PROGRAM PRG_04_SawAxes
VAR
	bUP						: BOOL;
	bDOWN					: BOOL;
	bCUT					: BOOL;
	bRETURN					: BOOL;
	
	bDoublePassCountUp		: BOOL;
	
	ctu_DoublePass			: CTU;
	
	iStep: INT;
	bUP_TON: TON;
//	bUP_TP: TP;
	rtrig1: r_trig;
//	ftrig1: f_trig;
	DoublePass_SR: SR;
	bDoublePassQ: BOOL;
	bUP_TON_IN: BOOL;
	autocrosscut_error: TON;
	RS_TriggerReturn: RS;
	RS_TriggerCUT: RS;
	R_TRIG_0: R_TRIG;
	R_TRIG_1: R_TRIG;
	R_TRIG_2: R_TRIG;
	R_TRIG_3: R_TRIG;
	R_TRIG_4: R_TRIG;
	R_TRIG_5: R_TRIG;
	RS_TriggerCUT2: RS;
	R_TRIG_10: R_TRIG;
	R_TRIG_11: R_TRIG;
	R_TRIG_12: R_TRIG;
	RS_TriggerReturn2: RS;
	R_TRIG_13: R_TRIG;
	R_TRIG_14: R_TRIG;
	R_TRIG_15: R_TRIG;

	rCutSpeed: REAL;
	rReturnSpeed: REAL;
	rVFDMaxSpeed: REAL;
	rBufferSpeed: REAL;
	rSawOFFSpeed: REAL;
	rSpeedScaled: REAL;
	// speed test
	iSpeedTest: INT;
	rSawCurrentTest: REAL;
	TON_step10: TON;
	TON_step20: TON;
	TON_step30: TON;
	TON_step40: TON;
	TON_step50: TON;
	TON_step60: TON;
	TON_DownDelay: TON;
END_VAR

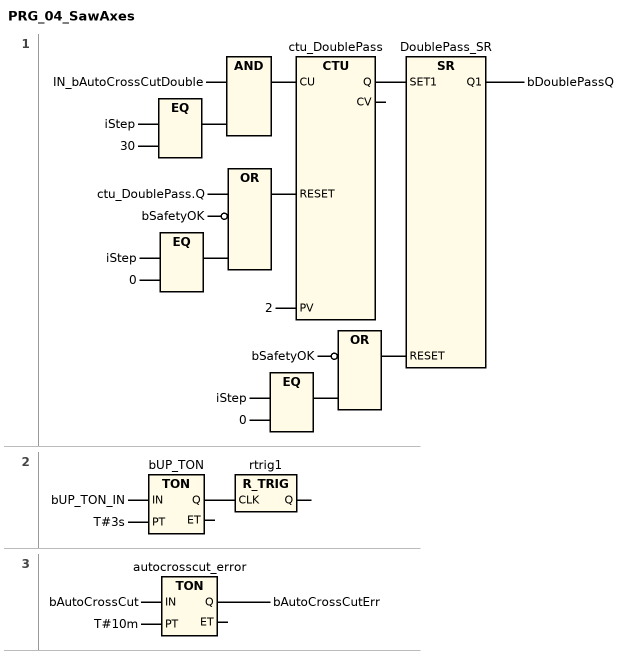
// NETWORK 1
ctu_DoublePass(
    CU := IN_bAutoCrossCutDouble AND iStep = 30,
    RESET := ctu_DoublePass.Q OR NOT bSafetyOK OR iStep = 0,
    PV := 2); // CTU
DoublePass_SR(SET1 := ctu_DoublePass.Q, RESET := NOT bSafetyOK OR iStep = 0); // SR
bDoublePassQ := DoublePass_SR.Q1;

// NETWORK 2
bUP_TON(IN := bUP_TON_IN, PT := T#3s); // TON
rtrig1(CLK := bUP_TON.Q); // R_TRIG

// NETWORK 3
autocrosscut_error(IN := bAutoCrossCut, PT := T#10m); // TON
bAutoCrossCutErr := autocrosscut_error.Q;

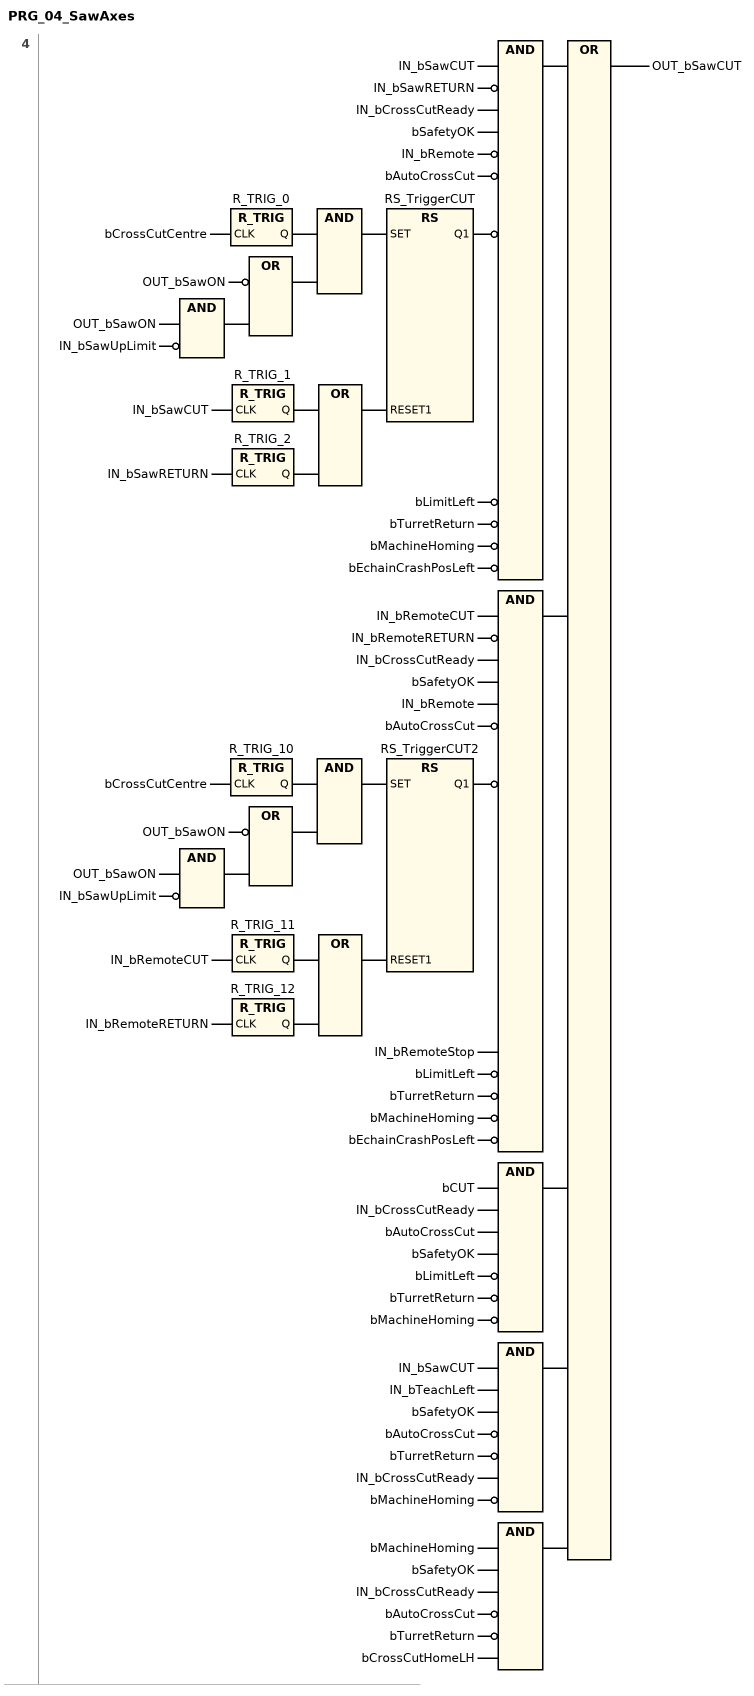
// NETWORK 4
R_TRIG_0(CLK := bCrossCutCentre); // R_TRIG
R_TRIG_1(CLK := IN_bSawCUT); // R_TRIG
R_TRIG_2(CLK := IN_bSawRETURN); // R_TRIG
RS_TriggerCUT(SET := R_TRIG_0.Q AND (NOT OUT_bSawON OR OUT_bSawON AND NOT IN_bSawUpLimit), RESET1 := R_TRIG_1.Q OR R_TRIG_2.Q); // RS
R_TRIG_10(CLK := bCrossCutCentre); // R_TRIG
R_TRIG_11(CLK := IN_bRemoteCUT); // R_TRIG
R_TRIG_12(CLK := IN_bRemoteRETURN); // R_TRIG
RS_TriggerCUT2(SET := R_TRIG_10.Q AND (NOT OUT_bSawON OR OUT_bSawON AND NOT IN_bSawUpLimit), RESET1 := R_TRIG_11.Q OR R_TRIG_12.Q); // RS
OUT_bSawCUT := IN_bSawCUT AND NOT IN_bSawRETURN AND IN_bCrossCutReady AND bSafetyOK AND NOT IN_bRemote AND NOT bAutoCrossCut AND NOT RS_TriggerCUT.Q1 AND NOT bLimitLeft AND NOT bTurretReturn AND NOT bMachineHoming AND NOT bEchainCrashPosLeft OR IN_bRemoteCUT AND NOT IN_bRemoteRETURN AND IN_bCrossCutReady AND bSafetyOK AND IN_bRemote AND NOT bAutoCrossCut AND NOT RS_TriggerCUT2.Q1 AND IN_bRemoteStop AND NOT bLimitLeft AND NOT bTurretReturn AND NOT bMachineHoming AND NOT bEchainCrashPosLeft OR bCUT AND IN_bCrossCutReady AND bAutoCrossCut AND bSafetyOK AND NOT bLimitLeft AND NOT bTurretReturn AND NOT bMachineHoming OR IN_bSawCUT AND IN_bTeachLeft AND bSafetyOK AND NOT bAutoCrossCut AND NOT bTurretReturn AND IN_bCrossCutReady AND NOT bMachineHoming OR bMachineHoming AND bSafetyOK AND IN_bCrossCutReady AND NOT bAutoCrossCut AND NOT bTurretReturn AND bCrossCutHomeLH;

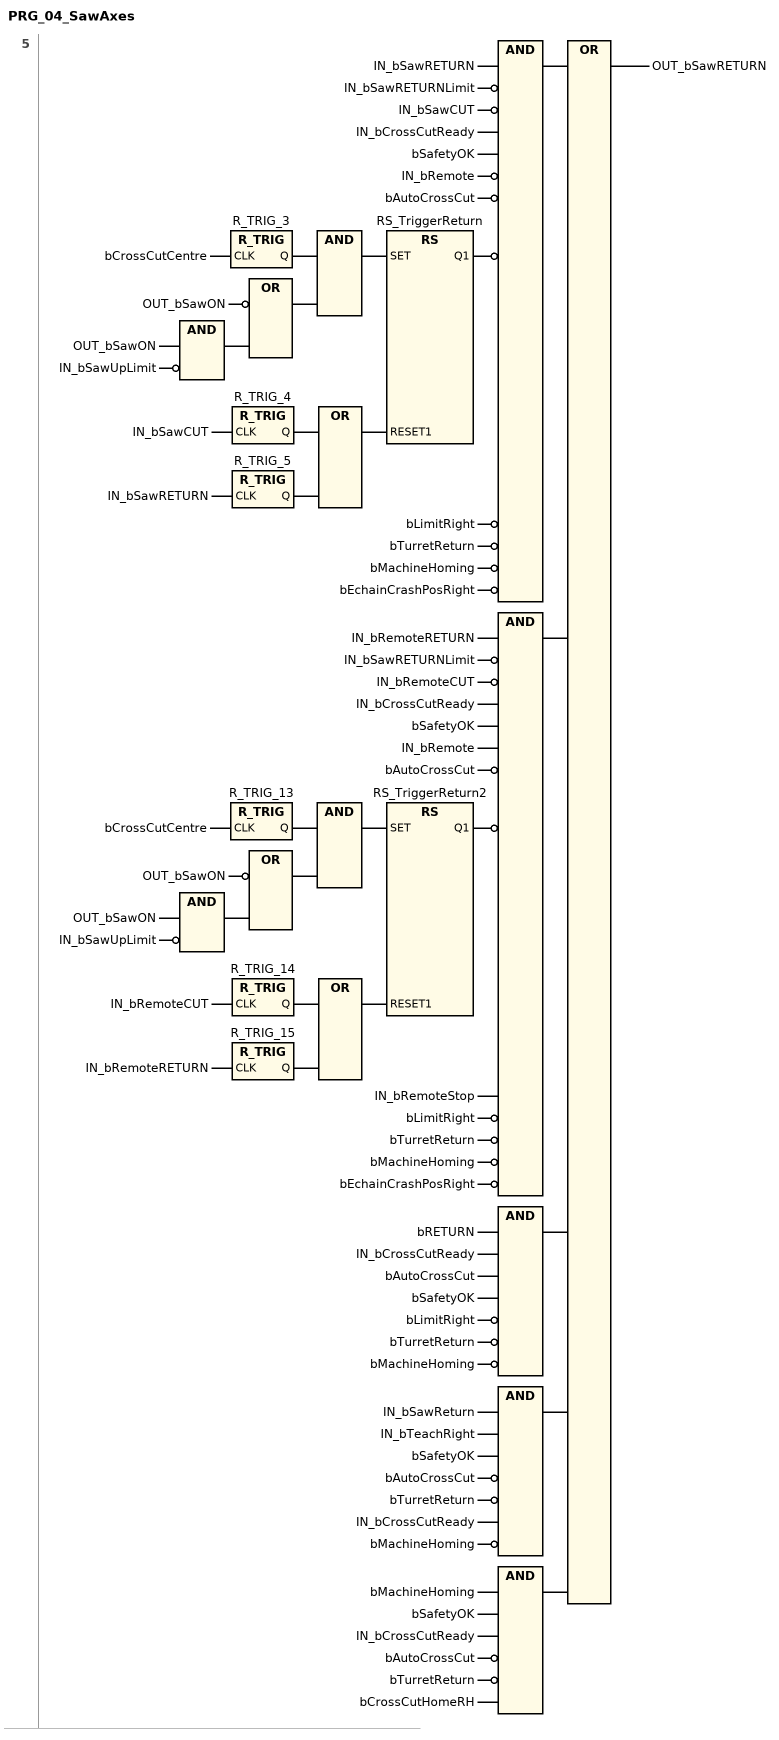
// NETWORK 5
R_TRIG_3(CLK := bCrossCutCentre); // R_TRIG
R_TRIG_4(CLK := IN_bSawCUT); // R_TRIG
R_TRIG_5(CLK := IN_bSawRETURN); // R_TRIG
RS_TriggerReturn(SET := R_TRIG_3.Q AND (NOT OUT_bSawON OR OUT_bSawON AND NOT IN_bSawUpLimit), RESET1 := R_TRIG_4.Q OR R_TRIG_5.Q); // RS
R_TRIG_13(CLK := bCrossCutCentre); // R_TRIG
R_TRIG_14(CLK := IN_bRemoteCUT); // R_TRIG
R_TRIG_15(CLK := IN_bRemoteRETURN); // R_TRIG
RS_TriggerReturn2(SET := R_TRIG_13.Q AND (NOT OUT_bSawON OR OUT_bSawON AND NOT IN_bSawUpLimit), RESET1 := R_TRIG_14.Q OR R_TRIG_15.Q); // RS
OUT_bSawRETURN := IN_bSawRETURN AND NOT IN_bSawRETURNLimit AND NOT IN_bSawCUT AND IN_bCrossCutReady AND bSafetyOK AND NOT IN_bRemote AND NOT bAutoCrossCut AND NOT RS_TriggerReturn.Q1 AND NOT bLimitRight AND NOT bTurretReturn AND NOT bMachineHoming AND NOT bEchainCrashPosRight OR IN_bRemoteRETURN AND NOT IN_bSawRETURNLimit AND NOT IN_bRemoteCUT AND IN_bCrossCutReady AND bSafetyOK AND IN_bRemote AND NOT bAutoCrossCut AND NOT RS_TriggerReturn2.Q1 AND IN_bRemoteStop AND NOT bLimitRight AND NOT bTurretReturn AND NOT bMachineHoming AND NOT bEchainCrashPosRight OR bRETURN AND IN_bCrossCutReady AND bAutoCrossCut AND bSafetyOK AND NOT bLimitRight AND NOT bTurretReturn AND NOT bMachineHoming OR IN_bSawReturn AND IN_bTeachRight AND bSafetyOK AND NOT bAutoCrossCut AND NOT bTurretReturn AND IN_bCrossCutReady AND NOT bMachineHoming OR bMachineHoming AND bSafetyOK AND IN_bCrossCutReady AND NOT bAutoCrossCut AND NOT bTurretReturn AND bCrossCutHomeRH;

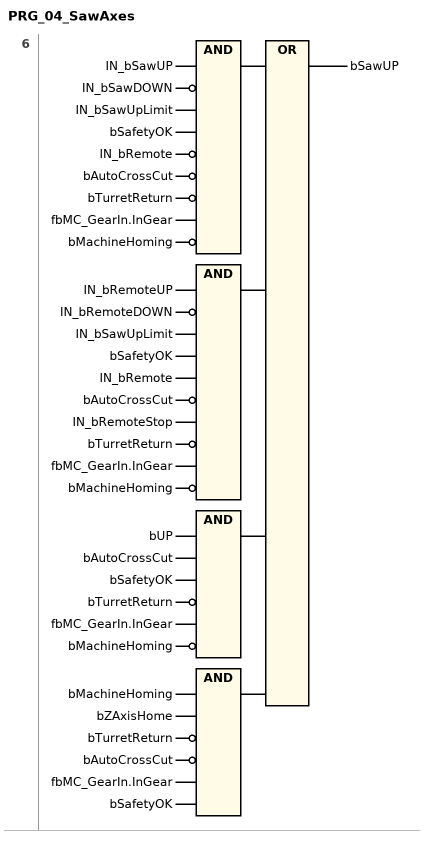
// NETWORK 6
bSawUP := IN_bSawUP AND NOT IN_bSawDOWN AND IN_bSawUpLimit AND bSafetyOK AND NOT IN_bRemote AND NOT bAutoCrossCut AND NOT bTurretReturn AND fbMC_GearIn.InGear AND NOT bMachineHoming OR IN_bRemoteUP AND NOT IN_bRemoteDOWN AND IN_bSawUpLimit AND bSafetyOK AND IN_bRemote AND NOT bAutoCrossCut AND IN_bRemoteStop AND NOT bTurretReturn AND fbMC_GearIn.InGear AND NOT bMachineHoming OR bUP AND bAutoCrossCut AND bSafetyOK AND NOT bTurretReturn AND fbMC_GearIn.InGear AND NOT bMachineHoming OR bMachineHoming AND bZAxisHome AND NOT bTurretReturn AND NOT bAutoCrossCut AND fbMC_GearIn.InGear AND bSafetyOK;

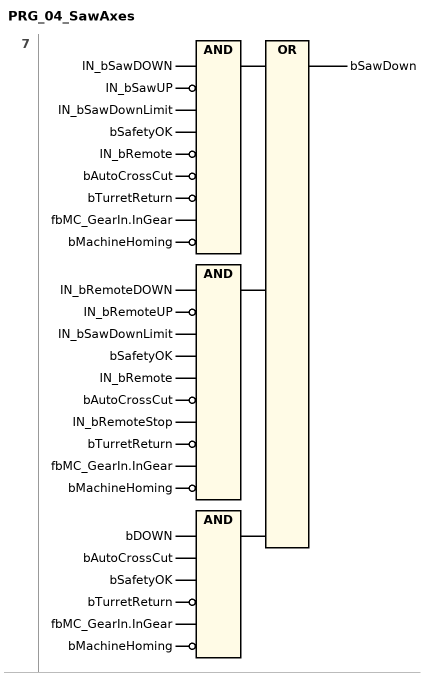
// NETWORK 7
bSawDown := IN_bSawDOWN AND NOT IN_bSawUP AND IN_bSawDownLimit AND bSafetyOK AND NOT IN_bRemote AND NOT bAutoCrossCut AND NOT bTurretReturn AND fbMC_GearIn.InGear AND NOT bMachineHoming OR IN_bRemoteDOWN AND NOT IN_bRemoteUP AND IN_bSawDownLimit AND bSafetyOK AND IN_bRemote AND NOT bAutoCrossCut AND IN_bRemoteStop AND NOT bTurretReturn AND fbMC_GearIn.InGear AND NOT bMachineHoming OR bDOWN AND bAutoCrossCut AND bSafetyOK AND NOT bTurretReturn AND fbMC_GearIn.InGear AND NOT bMachineHoming;

ACTION ACT_04_1_AutoCrossCut:
	IF		NOT bSafetyOK OR IN_FaultReset OR NOT OUT_bSawON
	THEN	iStep	:=	0;
	END_IF

	TON_DownDelay(IN:= , PT:= T#3S, Q=> , ET=> );
	IF		iStep <> 30 THEN
			TON_DownDelay.IN	:= FALSE ;
	END_IF
(* Double Pass counter BOOL *)
	IF		ctu_DoublePass.CV	=	1
	THEN	bDoublePassCountUp		:=	TRUE;
	ELSE	bDoublePassCountUp		:=	FALSE;
	END_IF

CASE iStep OF 
	0:		//	Step 0	:	Init step
				bAutoCrossCut	:= FALSE ;
				bUP				:= FALSE ;
				bDOWN			:= FALSE ;
				bCUT			:= FALSE ;
				bRETURN			:= FALSE ;
				bUP_TON_IN		:= FALSE ;
				
		IF
				bSafetyOK
				AND bTurret045Range
				AND OUT_bSawON
				AND (IN_bCrossCutLeft AND IN_bCrossCutRight AND NOT IN_bRemote)
				AND NOT (bTurretReturn OR bMachineHoming)
				AND NOT IN_bCarriageReference
		THEN
				bAutoCrossCut := TRUE	;
				iStep	:=		20		;
		ELSE
				bAutoCrossCut := FALSE	;
				iStep	:=		0		;
		END_IF

	20:		// Step 20	:	Saw RETURN movement
		IF 
				bAutoCrossCut
				AND bSafetyOK
				AND NOT bLimitRight
			
		THEN	bRETURN		:=	TRUE	;
		
		ELSE
				bRETURN		:=	FALSE	;
				iStep		:=	30		;
		END_IF
	
		IF 		NOT bSafetyOK
		THEN 	
				bRETURN		:=	FALSE	;
				iStep		:=	0		;
		END_IF
		
	30:		// Step 30	:	Saw DOWN movement
	ctu_DoublePass.CV;
		IF
				bAutoCrossCut
				AND bSafetyOK
				AND ((IN_bAutoCrossCutDouble AND IN_bDoublePassReference AND bDoublePassCountUp) 
					OR ( IN_bSawDownLimit AND (bDoublePassQ OR NOT bDoublePassCountUp)))
		THEN	
				bDOWN		:=	TRUE	;
		ELSE
				bDOWN		:=	FALSE	;
				TON_DownDelay.IN := TRUE ;
					IF TON_DownDelay.Q THEN
						iStep	:=	40		;
					END_IF
		END_IF
		
		IF 		NOT bSafetyOK
		THEN 	
				bDOWN		:=	FALSE	;
				iStep		:=	0		;
		END_IF
	
	40:		// Step 40	:	Saw CUT movement
		IF
				bAutoCrossCut
				AND bSafetyOK
				AND	NOT bLimitLeft
			THEN
				bCUT		:=	TRUE	;
		ELSE
				bCUT		:=	FALSE	;
				iStep		:=	50		;
		END_IF
		
		IF 		NOT bSafetyOK
			THEN 	
				bCUT		:=	FALSE	;
				iStep		:=	0		;
		END_IF
	
	50:		// Step 50	:	Saw UP movement		(* for double pass: only lift slightly, RETURN, then plunge all the way down *)
	ctu_DoublePass.CV;	
		IF
				IN_bAutoCrossCutDouble AND bDoublePassCountUp AND NOT bDoublePassQ
			THEN
				bUP_TON_IN	:=	TRUE	;
				bUP			:=	NOT bUP_TON.Q	;
				
				IF
					rtrig1.Q THEN
					iStep	:=	60	;
				END_IF
				
		ELSIF
				bAutoCrossCut
				AND bSafetyOK
				AND IN_bSawUpLimit
				AND ((bDoublePassQ AND NOT bDoublePassCountUp AND IN_bAutoCrossCutDouble) OR (NOT IN_bAutoCrossCutDouble))
			THEN
				bUP			:=	TRUE	;
		ELSE
				bUP			:=	FALSE	;
				iStep		:=	60		;
		END_IF
		
		IF 		NOT bSafetyOK
		THEN 	
				bUP			:=	FALSE	;
				iStep		:=	0		;
		END_IF
	
	60:		// Step 60	:	Saw RETURN movement (loop back to step 20 if double pass)
		IF
				IN_bAutoCrossCutDouble
				AND bDoublePassCountUp
		THEN
				iStep		:=	20		;
		ELSIF	
				bAutoCrossCut
				AND bSafetyOK
				AND NOT bCrossCutCentre
		THEN
				bRETURN		:=	TRUE	;
		ELSE
				bRETURN		:=	FALSE	;
				iStep		:=	0		;
		END_IF
	
END_CASE
END_ACTION

ACTION ACT_04_2_CrossCutSpeed:
// Cut and Return speed in VFD Hz
rCutSpeed := 5 ;
rReturnSpeed := 8.5 ;		
rVFDMaxSpeed := 20 ;		// set VFD P1-01 to this same Hz setting
rBufferSpeed := 2 ;
rSawOFFSpeed := 15 ;
rSpeedScaled := (INT_TO_REAL(OUT_iCrossCutFeedback) / 32767) * rVFDMaxSpeed ;
			
		IF fbSawCurrent.Out.rScaled < 40 THEN		// current feedback threshold
			rCrossCutSpeedMultiplier := 1 ;
		ELSIF fbSawCurrent.Out.rScaled > 40 AND fbSawCurrent.Out.rScaled < 55 THEN
			rCrossCutSpeedMultiplier := 0.75 ;
		ELSIF fbSawCurrent.Out.rScaled > 55 AND fbSawCurrent.Out.rScaled < 70 THEN
			rCrossCutSpeedMultiplier := 0.5 ;
		ELSIF fbSawCurrent.Out.rScaled > 70 AND fbSawCurrent.Out.rScaled < 85 THEN
			rCrossCutSpeedMultiplier := 0.4 ;
		ELSIF fbSawCurrent.Out.rScaled > 85 THEN
			rCrossCutSpeedMultiplier := 0.2 ;
		END_IF

IF OUT_bSawRETURN AND NOT OUT_bSawCUT AND NOT bApproachingLimitRight AND OUT_bSawON THEN	// Return speed if Saw blade is ON
	OUT_iCrossCutFeedback := REAL_TO_INT((rReturnSpeed / rVFDMaxSpeed) * 32767) ;
																	
ELSIF OUT_bSawCUT AND NOT OUT_bSawRETURN AND NOT bApproachingLimitLeft AND OUT_bSawON THEN	// Cut speed if Saw blade is ON
	OUT_iCrossCutFeedback := REAL_TO_INT(((rCutSpeed * rCrossCutSpeedMultiplier) / rVFDMaxSpeed) * 32767) ; // ##### CURRENT FEEDBACK #####
	
ELSIF ((OUT_bSawCUT AND bApproachingLimitLeft) OR (OUT_bSawRETURN AND bApproachingLimitRight))  THEN	// Buffer speed as the blade approaches the edge limits
	OUT_iCrossCutFeedback := REAL_TO_INT((rBufferSpeed / rVFDMaxSpeed) * 32767) ;
	
ELSIF ((OUT_bSawCUT AND NOT bApproachingLimitLeft) OR (OUT_bSawRETURN AND NOT bApproachingLimitRight)) AND NOT OUT_bSawON THEN // Cut and Return speed if Saw blade OFF
	OUT_iCrossCutFeedback := REAL_TO_INT((rSawOFFSpeed / rVFDMaxSpeed) * 32767) ;
ELSE
	OUT_iCrossCutFeedback := 0 ;
END_IF

(*		// Current Feedback Test
IF NOT bSafetyOK THEN
	iSpeedTest := 0;
END_IF

CASE iSpeedTest OF
	0: // 0 A before startup
		rSawCurrentTest := 0;
		TON_step10	.IN	:= FALSE ;
		TON_step20	.IN	:= FALSE ;
		TON_step30	.IN	:= FALSE ;
		TON_step40	.IN	:= FALSE ;
		TON_step50	.IN	:= FALSE ;
		TON_step60	.IN	:= FALSE ;
	10: // constant 33 A after startup for 3 sec
		TON_step10(IN:= , PT:= T#3S, Q=> , ET=> );
		TON_step10.IN := TRUE;
		rSawCurrentTest := 33;
		IF TON_step10.Q THEN
			iSpeedTest := 20;
		END_IF
	20: // increase to 38 A for 3 sec
		TON_step20(IN:= , PT:= T#3S, Q=> , ET=> );
		TON_step20.IN := TRUE;
		rSawCurrentTest := 38;
		IF TON_step20.Q THEN
			iSpeedTest := 30;
		END_IF
	30: // increase to 45 A for 2 sec
		TON_step30(IN:= , PT:= T#2S, Q=> , ET=> );
		TON_step30.IN := TRUE;
		rSawCurrentTest := 45;
		IF TON_step30.Q THEN
			iSpeedTest := 40;
		END_IF
	40: // decrease back to 38 A for 2 sec
		TON_step40(IN:= , PT:= T#2S, Q=> , ET=> );
		TON_step40.IN := TRUE;
		rSawCurrentTest := 38;
		IF TON_step40.Q THEN
			iSpeedTest := 50;
		END_IF
	50: // spike to 55 A for 0.5 sec
		TON_step50(IN:= , PT:= T#2S, Q=> , ET=> );
		TON_step50.IN := TRUE;
		rSawCurrentTest := 55;
		IF TON_step50.Q THEN
			iSpeedTest := 60;
		END_IF
	60: // decrease back to 38 A to finish the cut
		TON_step60(IN:= , PT:= T#2S, Q=> , ET=> );
		TON_step60.IN := TRUE;
		rSawCurrentTest := 38;
		IF TON_step60.Q THEN
			iSpeedTest := 0;
		END_IF
	
END_CASE
*)
END_ACTION

END_PROGRAM

(* stored: Version 1.1.0.1, ProductVersion 3.1.4024.12
   POU PRG_04_SawAxes: Id {abc17e14-5c43-41e6-8480-1dab67d5b81f}, SpecialFunc None
   Action ACT_04_1_AutoCrossCut: Id {37a29f44-dba5-4c4d-8257-7b5c2633111c}
   Action ACT_04_2_CrossCutSpeed: Id {c993172b-aa5a-4afa-9afe-d7df0835ca0b} *)
